(* IEC 61131-3 sources: AXOpen/src/components.rexroth.press/ctrl/src/AxoSmartFunctionKitDataTypes_v_4_x_x, 12 files *)

(* ---- eAxoSmartFunctionKitCommand_v_4_x_x.st ---- *)
NAMESPACE AXOpen.Components.Rexroth.Press
    TYPE PUBLIC
        eAxoSmartFunctionKitCommand_v_4_x_x : INT
        (
            StartProgram := 1,
            SetProgramActive := 2,
            Positioning := 3,
            Jog := 4,
            ClearError := 5,
            StopMovement := 6,
            RestartDrive := 7,
            Tare := 9,
            StartHoming := 10,
            SetSystemVariable := 11,
            LockParticipant := 12,
            SetReference := 13,
            ReadSystemVariable := 14
        );
    END_TYPE
END_NAMESPACE

(* ---- eAxoSmartFunctionKitParticipant_v_4_x_x.st ---- *)
NAMESPACE AXOpen.Components.Rexroth.Press
    TYPE PUBLIC
        eAxoSmartFunctionKitParticipant_v_4_x_x : INT
        (
            WebInterface := 1,
            Fieldbus := 2,
            PhysicalInputsOutputs := 3
        );
    END_TYPE
END_NAMESPACE

(* ---- eAxoSmartFunctionKitStatusInformation_v_4_x_x.st ---- *)
NAMESPACE AXOpen.Components.Rexroth.Press
    TYPE PUBLIC
        eAxoSmartFunctionKitStatusInformation_v_4_x_x : UINT
        (
            ActiveProgramNumber         := UINT#301, //  The PROGRAM number active in the drive is read out.
            RemainingStorageSpaceOnIPC  := UINT#302, // (PR21) The remaining storage space OF the IPC is transferred in MB.
            CurrentPosition             := UINT#401, //The cyclically transmitted position is read out.
            CurrentTravelSpeed          := UINT#402, // The cyclically transmitted travel speed is read out.
            CurrentForce                := UINT#403  // The cyclically transmitted force is read out
            );
    END_TYPE
END_NAMESPACE

(* ---- AxoSmartFunctionKit_ComponentStatus_v_4_x_x.st ---- *)
NAMESPACE AXOpen.Components.Rexroth.Press
    {S7.extern=ReadWrite}
    {#ix-attr:[Container(Layout.Stack)]}
    CLASS PUBLIC AxoSmartFunctionKit_ComponentStatus_v_4_x_x  EXTENDS AXOpen.Components.Abstractions.AxoComponent_Status
        VAR PUBLIC
            Status : AxoSmartFunctionKitStatus_v_4_x_x;
            {#ix-set:AttributeName = "<#Current command parameters#>"}
            CurrentCommandParameters : AxoSmartFunctionKitRequest_v_4_x_x;
        END_VAR
    END_CLASS
END_NAMESPACE

(* ---- AxoSmartFunctionKit_Config_v_4_x_x.st ---- *)
NAMESPACE AXOpen.Components.Rexroth.Press
    {#ix-attr:[Container(Layout.Stack)]}
    {S7.extern=ReadWrite}
    CLASS PUBLIC AxoSmartFunctionKit_Config_v_4_x_x
        VAR PUBLIC
            {#ix-set:AttributeName = "<#Info time#>"}
            InfoTime : LTIME := LT#10S;
            {#ix-set:AttributeName = "<#Error time#>"}
            ErrorTime : LTIME := LT#30S;
            {#ix-set:AttributeName = "<#Task timeout#>"}
            TaskTimeout : LTIME := LT#50S;
            {#ix-set:AttributeName = "<#Location of the curve export#>"}
            CurveExportLocation : STRING ;
            {#ix-set:AttributeName = "<#Ip address#>"}
            IpAddress : STRING ;
        END_VAR
    END_CLASS
END_NAMESPACE

(* ---- AxoSmartFunctionKit_Control_v_4_x_x.st ---- *)
NAMESPACE AXOpen.Components.Rexroth.Press
    {S7.extern=ReadWrite}
    {#ix-attr:[Container(Layout.Wrap)]}
    CLASS AxoSmartFunctionKit_Control_v_4_x_x
        VAR PUBLIC
            {#ix-attr:[Container(Layout.Stack)]}
            {#ix-attr:[Group(GroupLayout.GroupBox)]}
            {#ix-set:AttributeName = "<#Handle#>"}
            Handle                  : WORD;
            {#ix-set:AttributeName = "<#Command#>"}
            Command                  : WORD;
            {#ix-set:AttributeName = "<#Value 1#>"}
            Value1                  : DWORD;
            {#ix-set:AttributeName = "<#Value 2#>"}
            Value2                  : DWORD;
            {#ix-set:AttributeName = "<#Value 3#>"}
            Value3                  : DWORD;
            {#ix-set:AttributeName = "<#Value 4#>"}
            Value4                  : DWORD;
            {#ix-set:AttributeName = "<#Value 5#>"}
            Value5                  : DWORD;
            {#ix-set:AttributeName = "<#Value 6#>"}
            Value6                  : DWORD;
            {#ix-set:AttributeName = "<#Value 7#>"}
            Value7                  : DWORD;
            {#ix-set:AttributeName = "<#Virtual Io#>"}
            VirtualIo               : WORD;
            {#ix-set:AttributeName = "<#Fast variable control#>"}
            FastVarControl	        : DWORD;
            {#ix-set:AttributeName = "<#Fast variable data#>"}
            FastVarData	            : DWORD;
        END_VAR
    END_CLASS
END_NAMESPACE

(* ---- AxoSmartFunctionKit_HWIDs_v_4_x_x.st ---- *)
NAMESPACE AXOpen.Components.Rexroth.Press
   {S7.extern=ReadWrite}
	CLASS AxoSmartFunctionKit_HWIDs_v_4_x_x
      VAR PUBLIC
         {#ix-set:AttributeName = "<#Hardware ID Device#>"}
         HW_Device            : UINT;
         {#ix-set:AttributeName = "<#Hardware ID 'ParamCh_IDN' module#>"}
         HW_ParamCh_IDN           : UINT;
         {#ix-set:AttributeName = "<#Hardware ID 'F_ModulNotUsed' module#>"}
         HW_F_ModulNotUsed            : UINT;
         {#ix-set:AttributeName = "<#Hardware ID 'Input_24_Words' submodule#>"}
         HW_Input_24_Words      : UINT;
         {#ix-set:AttributeName = "<#Hardware ID 'Output_21_Words' submodule#>"}
         HW_Output_21_Words      : UINT;
      END_VAR
   END_CLASS
END_NAMESPACE

(* ---- AxoSmartFunctionKit_State_v_4_x_x.st ---- *)
NAMESPACE AXOpen.Components.Rexroth.Press
    {S7.extern=ReadWrite}
    {#ix-attr:[Container(Layout.Wrap)]}
    CLASS AxoSmartFunctionKit_State_v_4_x_x
        VAR PUBLIC
            {#ix-attr:[Container(Layout.Stack)]}
            {#ix-attr:[Group(GroupLayout.GroupBox)]}
            {#ix-set:AttributeName = "<#Handle#>"}
            Handle                  : WORD;
            {#ix-set:AttributeName = "<#Status#>"}
            Status                  : WORD;
            {#ix-set:AttributeName = "<#Value1#>"}
            Value1                  : DWORD;
            {#ix-set:AttributeName = "<#Value2#>"}
            Value2                  : DWORD;
            {#ix-set:AttributeName = "<#Value3#>"}
            Value3                  : DWORD;
            {#ix-set:AttributeName = "<#NotificationId#>"}
            NotificationId          : WORD;
            {#ix-set:AttributeName = "<#NotificationValue#>"}
            NotificationValue       : DWORD;
            {#ix-set:AttributeName = "<#NotificationStatus#>"}
            NotificationStatus      : WORD;
            {#ix-set:AttributeName = "<#NotificationPosition#>"}
            NotificationPosition    : DWORD;
            {#ix-set:AttributeName = "<#NotificationVelocity#>"}
            NotificationVelocity    : DWORD;
            {#ix-set:AttributeName = "<#NotificationForce#>"}
            NotificationForce       : DWORD;
            {#ix-set:AttributeName = "<#DigitalIoMapping#>"}
            DigitalIoMapping        : WORD;
            {#ix-set:AttributeName = "<#VirtualIo#>"}
            VirtualIo               : WORD;
            {#ix-set:AttributeName = "<#Fast variable state#>"}
            FastVarState	        : DWORD;
            {#ix-set:AttributeName = "<#Fast variable data#>"}
            FastVarData	            : DWORD;
        END_VAR
    END_CLASS
END_NAMESPACE

(* ---- AxoSmartFunctionKitResponse_v_4_x_x.st ---- *)
NAMESPACE AXOpen.Components.Rexroth.Press
    {#ix-attr:[Container(Layout.Stack)]}
    {S7.extern=ReadWrite}
    CLASS PUBLIC AxoSmartFunctionKitResponse_v_4_x_x
        VAR PUBLIC
            {#ix-set:AttributeName = "<#Axis in reference#>"}
            AxisInReference : BOOL;
            {#ix-set:AttributeName = "<#Program active#>"}
            ProgramActive : BOOL;
            {#ix-set:AttributeName = "<#Last pressing Ok#>"}
            LastPressingOk : BOOL;
            {#ix-set:AttributeName = "<#Last pressing Nok#>"}
            LastPressingNok : BOOL;
            {#ix-set:AttributeName = "<#Sensor tared#>"}
            SensorTared : BOOL;
            {#ix-set:AttributeName = "<#Press ready#>"}
            PressReady : BOOL;
            {#ix-set:AttributeName = "<#Error#>"}
            Error : BOOL;
            {#ix-set:AttributeName = "<#Warning#>"}
            Warning : BOOL;
            {#ix-set:AttributeName = "<#Request possible#>"}
            RequestPossible : BOOL;
            {#ix-set:AttributeName = "<#Respons avialable#>"}
            ResponsAvialable : BOOL;
            {#ix-set:AttributeName = "<#Notification available#>"}
            NotificationAvailable : BOOL;
            {#ix-set:AttributeName = "<#Emergency off active#>"}
            EmergencyOffActive : BOOL;
            {#ix-set:AttributeName = "<#Safe standstill active#>"}
            SafeStandstillActive : BOOL;
        END_VAR
    END_CLASS
END_NAMESPACE

(* ---- AxoSmartFunctionKitResults_v_4_x_x.st ---- *)
NAMESPACE AXOpen.Components.Rexroth.Press
    {#ix-attr:[Container(Layout.Stack)]}
    {S7.extern=ReadWrite}
    CLASS PUBLIC AxoSmartFunctionKitResults_v_4_x_x
        VAR PUBLIC
            {#ix-set:AttributeName = "<#Id#>"}
            id : STRING;
            {#ix-set:AttributeName = "<#Maximal force#>"}
            maxForce : REAL;
            {#ix-set:AttributeName = "<#Maximal position#>"}
            maxPosition : REAL;
            {#ix-set:AttributeName = "<#Valid#>"}
            valid : BOOL;
            {#ix-set:AttributeName = "<#Creation date#>"}
            createdDate : DATE_AND_TIME;
            {#ix-set:AttributeName = "<#Cycle time#>"}
            cycleTime : REAL;
            {#ix-set:AttributeName = "<#Validation time#>"}
            validationTime : INT;
            {#ix-set:AttributeName = "<#Status#>"}
            status : STRING;
            {#ix-set:AttributeName = "<#Custom Id#>"}
            customId : STRING;
            {#ix-set:AttributeName = "<#Data recording disabled#>"}
            dataRecordingDisabled : BOOL;
            {#ix-set:AttributeName = "<#Sampling interval#>"}
            samplingInterval : INT;
            {#ix-set:AttributeName = "<#_v#>"}
            _v : INT;
        END_VAR
    END_CLASS
END_NAMESPACE

(* ---- AxoSmartFunctionKitStatus_v_4_x_x.st ---- *)
NAMESPACE AXOpen.Components.Rexroth.Press
    {#ix-attr:[Container(Layout.Stack)]}
    {S7.extern=ReadWrite}
    CLASS PUBLIC AxoSmartFunctionKitStatus_v_4_x_x
        VAR PUBLIC
            {#ix-set:AttributeName = "<#Response status#>"}
            ResponseStatus : AxoSmartFunctionKitResponse_v_4_x_x;
            {#ix-set:AttributeName = "<#Notification Id#>"}
            NotificationId  : UINT;
            {#ix-set:AttributeName = "<#Notification to display#>"}
            NotificationToDisplay  : eAxoSmartFunctionKitStatusInformation_v_4_x_x;
            {#ix-set:AttributeName = "<#Notification position#>"}
            NotificationPosition  : REAL;
            {#ix-set:AttributeName = "<#Notification velocity#>"}
            NotificationVelocity : REAL;
            {#ix-set:AttributeName = "<#Notification force#>"}
            NotificationForce : REAL;
            {#ix-set:AttributeName = "<#Digital Io mapping#>"}
            DigitalIoMapping : DWORD;
            {#ix-set:AttributeName = "<#Virtual Io#>"}
            VirtualIo  : DWORD;
        END_VAR
    END_CLASS
END_NAMESPACE

(* ---- AxoSmartFunctionKitRequest_v_4_x_x.st ---- *)
NAMESPACE AXOpen.Components.Rexroth.Press
    // {#ix-attr:[Container(Layout.Stack)]}
    // {S7.extern=ReadWrite}
    // CLASS PUBLIC AxoSmartFunctionKitRequest_v_4_x_x
    //     VAR PUBLIC
    TYPE AxoSmartFunctionKitRequest_v_4_x_x :
        STRUCT
            {#ix-set:AttributeName = "<#Command#>"}
            Command : eAxoSmartFunctionKitCommand_v_4_x_x;
            {#ix-set:AttributeName = "<#Serial number#>"}
            SerialNumber:STRING[28];
            {#ix-set:AttributeName = "<#Program Id#>"}
            ProgramId:INT;
            {#ix-set:AttributeName = "<#Position distance tara#>"}
            PositionDistanceTara:REAL;
            {#ix-set:AttributeName = "<#Travel speed#>"}
            TravelSpeed:REAL;
            {#ix-set:AttributeName = "<#Acceleration#>"}
            Acceleration:REAL;
            {#ix-set:AttributeName = "<#Offset#>"}
            Offset:REAL;
        END_STRUCT;
    END_TYPE

            // {#ix-set:AttributeName = "<#Value 1#>"}
            // Value1:DWORD;
            // {#ix-set:AttributeName = "<#Value 2#>"}
            // Value2:DWORD;
            // {#ix-set:AttributeName = "<#Value 3#>"}
            // Value3:DWORD;
            // {#ix-set:AttributeName = "<#Value 4#>"}
            // Value4:DWORD;
            // {#ix-set:AttributeName = "<#Value 5#>"}
            // Value5:DWORD;
            // {#ix-set:AttributeName = "<#Value 6#>"}
            // Value6:DWORD;
            // {#ix-set:AttributeName = "<#Value 7#>"}
            // Value7:DWORD;
    //     END_VAR
    // END_CLASS
END_NAMESPACE
